SUBAPPLICATION AX_SoftkeyToggle_RS_TO_AX (* Toggle-Trigger (SoftKey ODER AUX ODER lokale Web-/Dashboard-Methode ODER IO-Diag-Testbutton, via Softkey_Aux_Method_Button_IE) und Reset-Trigger (SoftKey ODER AUX ODER lokale Web-/Dashboard-Methode, via Softkey_Aux_Method_IE) treiben einen reinen AX-Zustand (AX_T_FF_SR.Q) - KEIN physischer Ausgang, KEINE Hintergrundfarbe, KEIN State-Publish. Basis-Baustein: fuer 1 Ausgang MyLib::sys::AX_SoftkeyToggle_RS_TO_QXA_BG (wrapt diesen Baustein), fuer mehrere zeitversetzte Ausgaenge (z.B. Baender-Sequenzierung) diesen Baustein direkt verwenden und den OUT-Zustand selbst mit AX_TON/AX_TOF pro Kanal weiterverarbeiten. *)
  (* Standard: 61499-2; Description: Copyright (c) 2026 Meisterschulen am Ostbahnhof This program and the accompanying materials are made available under the terms of the Eclipse Public License 2.0 which is available at https://www.eclipse.org/legal/epl-2.0/ SPDX-License-Identifier: EPL-2.0 *)
  (* Version 1.4, 2026-09-16, Franz Höpfinger, Meisterschulen am Ostbahnhof, Event-Input RESET in AUS umbenannt (Franz: 'der Eingang soll AUS heissen') - Namenskonsistenz mit Baender_Individual_Toggle/Baender_EinAus/Aufnahme_Automatik/Ernteseite_Antriebe, die alle denselben zentralen 'Alles Aus'-Softkey verteilen. *)
  (* Version 1.3, 2026-09-16, Franz Höpfinger, Meisterschulen am Ostbahnhof, Event-Input RESET ergaenzt (rein additiv, zusaetzlich zum bestehenden Reset.IND-Pfad auf AX_T_FF_SR.R verdrahtet) - fuer einen zentral gelesenen, gemeinsamen SoftKey (z.B. 'Alles Aus'), der mehrere Toggle-Instanzen gleichzeitig per Event zuruecksetzen soll, statt dass jede Instanz denselben SoftKey/AuxFunction2 nochmal einzeln selbst liest. *)
  (* Version 1.2, 2026-09-15, Franz Höpfinger, Meisterschulen am Ostbahnhof, FORCE_OFF Socket (AX) ergaenzt - analog Automatik_Toggle_Button.FORCE_OFF: steigende Flanke (AX_R_TRIG) resettet AX_T_FF_SR zusaetzlich zum bestehenden VT-Reset. Fuer eine uebergeordnete Sicherheitsabschaltung (z.B. Zapfwelle_Ueberwachung, KVE14 Zeile 33) - rein additiv, bestehende Instanzen muessen den neuen Socket verdrahten (z.B. auf einen festen FALSE-Literal, wenn nicht gebraucht). *)
  (* Version 1.1, 2026-09-15, Franz Höpfinger, Meisterschulen am Ostbahnhof, Toggle.u16ObjId_TEST -> Toggle.u16ObjIdB nachgezogen (Softkey_Aux_Method_Button_IE v1.1: u16ObjId_TEST dort auf u16ObjIdB umbenannt). Eigenes u16ObjId_TEST bleibt unveraendert. *)
  PACKAGE MyLib::sys;
  IMPORT isobus::UT::Q::const::IDs::ID_NULL;
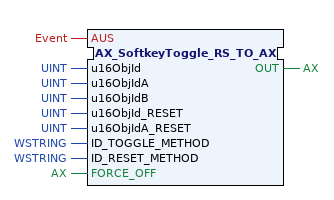
  EVENT_INPUT
    AUS; (* Reset hart auf AUS, von aussen als Event (z.B. 1 zentral gelesener gemeinsamer SoftKey) - zusaetzlich zum eigenen u16ObjId_RESET/u16ObjIdA_RESET/ID_RESET_METHOD-Pfad. Unverdrahtet lassen, wenn nicht gebraucht. *)
  END_EVENT
  VAR_INPUT
    u16ObjId : UINT := ID_NULL; (* Object ID Softkey Ein/Aus (Toggle) *)
    u16ObjIdA : UINT := ID_NULL; (* Object ID AuxFunction2 (Joystick) fuer den Toggle - gleichberechtigt zum SoftKey *)
    u16ObjIdB : UINT := ID_NULL; (* Object ID IO-Diag-Testbutton (Ausgaenge-Diagnoseseite) - toggelt gleichberechtigt mit. ID_NULL lassen, wenn kein IO-Diag-Testbutton an diesem Toggle beteiligt sein soll *)
    u16ObjId_RESET : UINT := ID_NULL; (* Object ID Softkey 'Alles Aus' (Reset, hart auf AUS) - z.B. SoftKey_AUS *)
    u16ObjIdA_RESET : UINT := ID_NULL; (* Object ID AuxFunction2 (Joystick) fuer den Reset - gleichberechtigt zum Softkey 'Alles Aus' *)
    ID_TOGGLE_METHOD : WSTRING; (* Lokale Methodenadresse (ACTION=CREATE_METHOD) fuer den argumentlosen Toggle-Trigger - wird von Web-Client (vt-ui-mirror) UND direkt vom OPC-Dashboard aufgerufen *)
    ID_RESET_METHOD : WSTRING; (* Lokale Methodenadresse (ACTION=CREATE_METHOD) fuer den argumentlosen Reset-Trigger (hart auf AUS) - wird von Web-Client UND OPC-Dashboard aufgerufen *)
  END_VAR
  SOCKETS
    FORCE_OFF : adapter::types::unidirectional::AX; (* Optional: steigende Flanke resettet hart auf AUS (z.B. Sicherheitsabschaltung). Unverdrahtet lassen (fester FALSE-Literal), wenn nicht gebraucht. *)
  END_SOCKETS
  PLUGS
    OUT : adapter::types::unidirectional::AX; (* Toggle-Zustand (AX_T_FF_SR.Q) - Weiterverarbeitung (Ausgang, Hintergrund, Verzoegerung) bleibt dem Aufrufer ueberlassen *)
  END_PLUGS
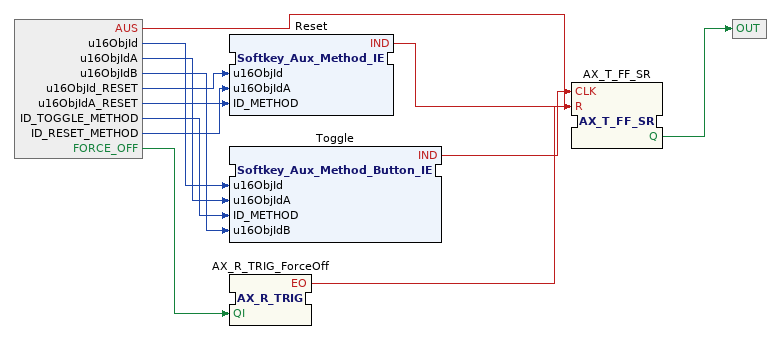
  (* AX_T_FF_SR.Q ist die EINZIGE Source of Truth - Toggle (SoftKey+AUX+Web/Dashboard-Methode+IO-Diag-Testbutton) und Reset (SoftKey+AUX+Web/Dashboard-Methode) sind alle reine argumentlose Event-Trigger - keine gemeinsame Variable. *)
  FBS
    AX_T_FF_SR : adapter::events::unidirectional::AX_T_FF_SR;
    AX_R_TRIG_ForceOff : adapter::events::unidirectional::AX_R_TRIG;
  END_FBS
  SUBAPPS
    Toggle : MyLib::sys::Softkey_Aux_Method_Button_IE;
    Reset : MyLib::sys::Softkey_Aux_Method_IE;
  END_SUBAPPS
  EVENT_CONNECTIONS
    Toggle.IND TO AX_T_FF_SR.CLK;
    Reset.IND TO AX_T_FF_SR.R;
    AX_R_TRIG_ForceOff.EO TO AX_T_FF_SR.R;
    AUS TO AX_T_FF_SR.R;
  END_CONNECTIONS
  DATA_CONNECTIONS
    u16ObjId TO Toggle.u16ObjId;
    u16ObjIdA TO Toggle.u16ObjIdA;
    ID_TOGGLE_METHOD TO Toggle.ID_METHOD;
    u16ObjIdB TO Toggle.u16ObjIdB;
    u16ObjId_RESET TO Reset.u16ObjId;
    u16ObjIdA_RESET TO Reset.u16ObjIdA;
    ID_RESET_METHOD TO Reset.ID_METHOD;
  END_CONNECTIONS
  ADAPTER_CONNECTIONS
    AX_T_FF_SR.Q TO OUT;
    FORCE_OFF TO AX_R_TRIG_ForceOff.QI;
  END_CONNECTIONS
END_SUBAPPLICATION
